(* Manuals for all controls to be used on the HMI
	rules 
		manuals are of type bool or HMI_PB_Safe
		manuals are reset when leaving manual_K (this is already implemented in SCM_Template)
		manuals are only used for manual stuff (see previous point why you can't do anything else with it)
*)
TYPE HMI_MAN :
STRUCT
	{info 'TODO TEMPLATE REMOVE: Example scam'}
	Example:HMI_MAN_TemplateMachinePart; 					//Example for how to use, remove me
END_STRUCT
END_TYPE

(* stored: Version 1.1.0.1, ProductVersion 3.1.4024.12
   DUT HMI_MAN: Id {642aac16-8a42-4b1e-bf0d-b824f6d2c325} *)
